PROGRAM P1_03_Alarms
VAR
	i					:USINT;
	bAlarmActive		:BOOL;
	bAlarmDisabled		:BOOL;
	TON_AlarmOK			:TON;

END_VAR
VAR PERSISTENT
	fbAlarm				:ARRAY [0..69] OF FB_AlarmDiagnostic;
END_VAR

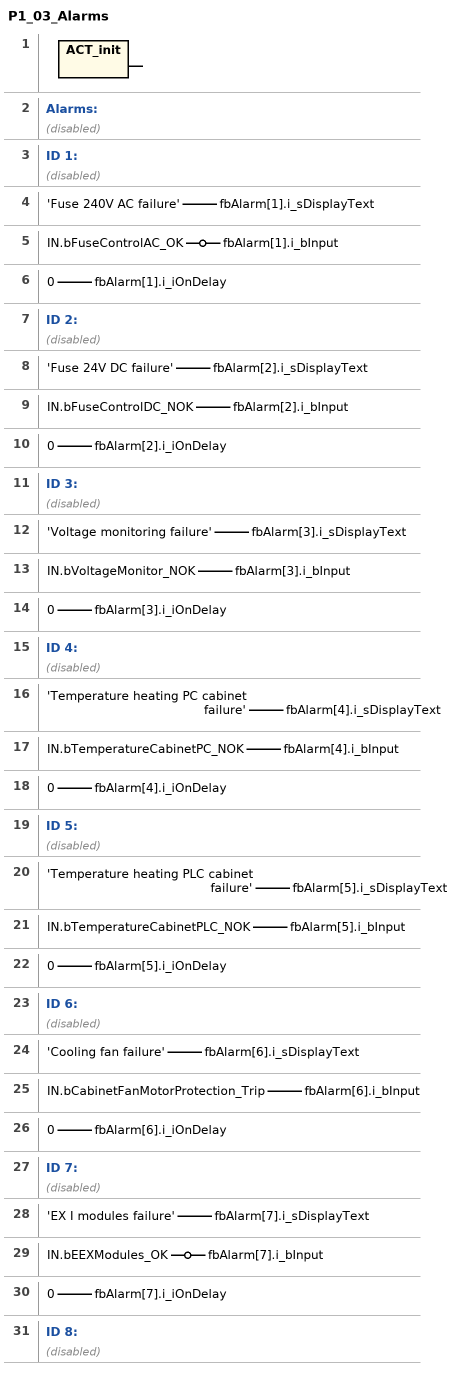
// NETWORK 1
ACT_init();

// NETWORK 2 (disabled)
// label: Alarms

// NETWORK 3 (disabled)
// label: ID 1

// NETWORK 4
fbAlarm[1].i_sDisplayText := 'Fuse 240V AC failure';

// NETWORK 5
fbAlarm[1].i_bInput := NOT IN.bFuseControlAC_OK;

// NETWORK 6
fbAlarm[1].i_iOnDelay := 0;

// NETWORK 7 (disabled)
// label: ID 2

// NETWORK 8
fbAlarm[2].i_sDisplayText := 'Fuse 24V DC failure';

// NETWORK 9
fbAlarm[2].i_bInput := IN.bFuseControlDC_NOK;

// NETWORK 10
fbAlarm[2].i_iOnDelay := 0;

// NETWORK 11 (disabled)
// label: ID 3

// NETWORK 12
fbAlarm[3].i_sDisplayText := 'Voltage monitoring failure';

// NETWORK 13
fbAlarm[3].i_bInput := IN.bVoltageMonitor_NOK;

// NETWORK 14
fbAlarm[3].i_iOnDelay := 0;

// NETWORK 15 (disabled)
// label: ID 4

// NETWORK 16
fbAlarm[4].i_sDisplayText := 'Temperature heating PC cabinet failure';

// NETWORK 17
fbAlarm[4].i_bInput := IN.bTemperatureCabinetPC_NOK;

// NETWORK 18
fbAlarm[4].i_iOnDelay := 0;

// NETWORK 19 (disabled)
// label: ID 5

// NETWORK 20
fbAlarm[5].i_sDisplayText := 'Temperature heating PLC cabinet failure';

// NETWORK 21
fbAlarm[5].i_bInput := IN.bTemperatureCabinetPLC_NOK;

// NETWORK 22
fbAlarm[5].i_iOnDelay := 0;

// NETWORK 23 (disabled)
// label: ID 6

// NETWORK 24
fbAlarm[6].i_sDisplayText := 'Cooling fan failure';

// NETWORK 25
fbAlarm[6].i_bInput := IN.bCabinetFanMotorProtection_Trip;

// NETWORK 26
fbAlarm[6].i_iOnDelay := 0;

// NETWORK 27 (disabled)
// label: ID 7

// NETWORK 28
fbAlarm[7].i_sDisplayText := 'EX I modules failure';

// NETWORK 29
fbAlarm[7].i_bInput := NOT IN.bEEXModules_OK;

// NETWORK 30
fbAlarm[7].i_iOnDelay := 0;

// NETWORK 31 (disabled)
// label: ID 8

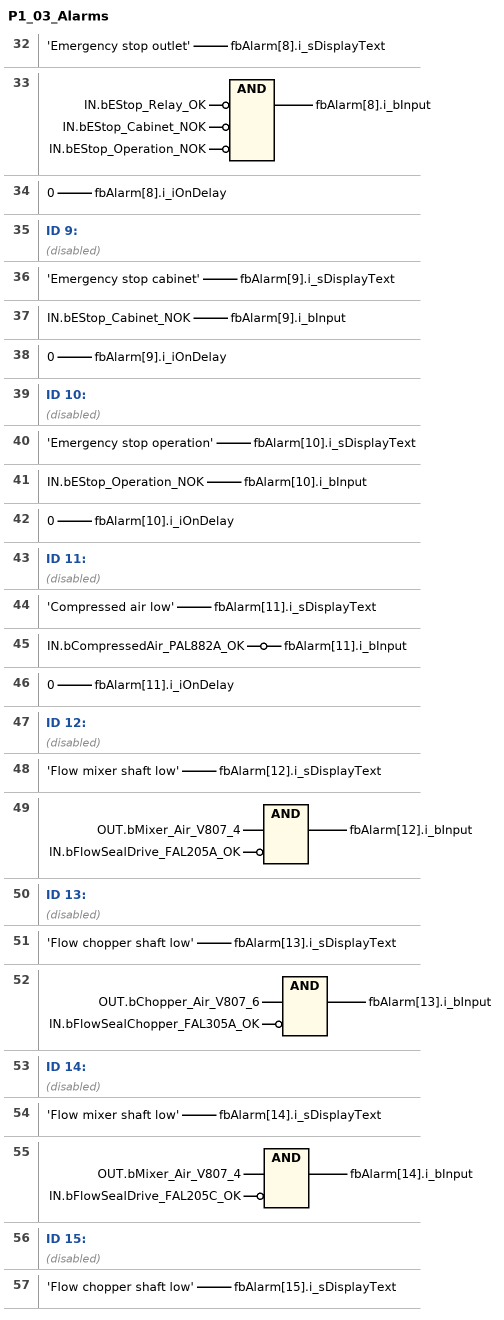
// NETWORK 32
fbAlarm[8].i_sDisplayText := 'Emergency stop outlet';

// NETWORK 33
fbAlarm[8].i_bInput := NOT IN.bEStop_Relay_OK AND NOT IN.bEStop_Cabinet_NOK AND NOT IN.bEStop_Operation_NOK;

// NETWORK 34
fbAlarm[8].i_iOnDelay := 0;

// NETWORK 35 (disabled)
// label: ID 9

// NETWORK 36
fbAlarm[9].i_sDisplayText := 'Emergency stop cabinet';

// NETWORK 37
fbAlarm[9].i_bInput := IN.bEStop_Cabinet_NOK;

// NETWORK 38
fbAlarm[9].i_iOnDelay := 0;

// NETWORK 39 (disabled)
// label: ID 10

// NETWORK 40
fbAlarm[10].i_sDisplayText := 'Emergency stop operation';

// NETWORK 41
fbAlarm[10].i_bInput := IN.bEStop_Operation_NOK;

// NETWORK 42
fbAlarm[10].i_iOnDelay := 0;

// NETWORK 43 (disabled)
// label: ID 11

// NETWORK 44
fbAlarm[11].i_sDisplayText := 'Compressed air low';

// NETWORK 45
fbAlarm[11].i_bInput := NOT IN.bCompressedAir_PAL882A_OK;

// NETWORK 46
fbAlarm[11].i_iOnDelay := 0;

// NETWORK 47 (disabled)
// label: ID 12

// NETWORK 48
fbAlarm[12].i_sDisplayText := 'Flow mixer shaft low';

// NETWORK 49
fbAlarm[12].i_bInput := OUT.bMixer_Air_V807_4 AND NOT IN.bFlowSealDrive_FAL205A_OK;

// NETWORK 50 (disabled)
// label: ID 13

// NETWORK 51
fbAlarm[13].i_sDisplayText := 'Flow chopper shaft low';

// NETWORK 52
fbAlarm[13].i_bInput := OUT.bChopper_Air_V807_6 AND NOT IN.bFlowSealChopper_FAL305A_OK;

// NETWORK 53 (disabled)
// label: ID 14

// NETWORK 54
fbAlarm[14].i_sDisplayText := 'Flow mixer shaft low';

// NETWORK 55
fbAlarm[14].i_bInput := OUT.bMixer_Air_V807_4 AND NOT IN.bFlowSealDrive_FAL205C_OK;

// NETWORK 56 (disabled)
// label: ID 15

// NETWORK 57
fbAlarm[15].i_sDisplayText := 'Flow chopper shaft low';

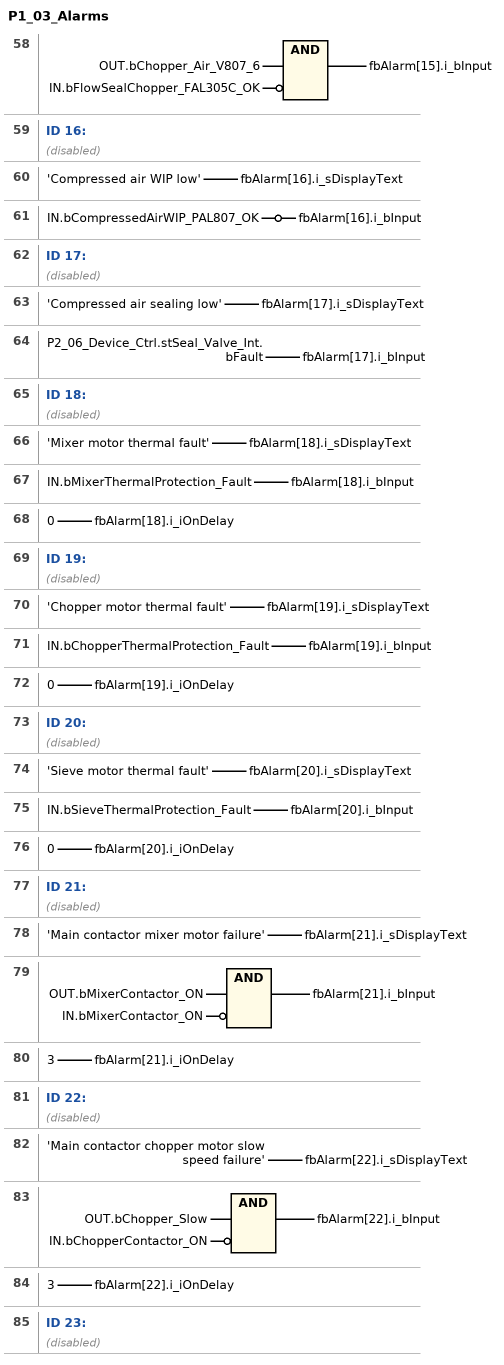
// NETWORK 58
fbAlarm[15].i_bInput := OUT.bChopper_Air_V807_6 AND NOT IN.bFlowSealChopper_FAL305C_OK;

// NETWORK 59 (disabled)
// label: ID 16

// NETWORK 60
fbAlarm[16].i_sDisplayText := 'Compressed air WIP low';

// NETWORK 61
fbAlarm[16].i_bInput := NOT IN.bCompressedAirWIP_PAL807_OK;

// NETWORK 62 (disabled)
// label: ID 17

// NETWORK 63
fbAlarm[17].i_sDisplayText := 'Compressed air sealing low';

// NETWORK 64
fbAlarm[17].i_bInput := P2_06_Device_Ctrl.stSeal_Valve_Int.bFault;

// NETWORK 65 (disabled)
// label: ID 18

// NETWORK 66
fbAlarm[18].i_sDisplayText := 'Mixer motor thermal fault';

// NETWORK 67
fbAlarm[18].i_bInput := IN.bMixerThermalProtection_Fault;

// NETWORK 68
fbAlarm[18].i_iOnDelay := 0;

// NETWORK 69 (disabled)
// label: ID 19

// NETWORK 70
fbAlarm[19].i_sDisplayText := 'Chopper motor thermal fault';

// NETWORK 71
fbAlarm[19].i_bInput := IN.bChopperThermalProtection_Fault;

// NETWORK 72
fbAlarm[19].i_iOnDelay := 0;

// NETWORK 73 (disabled)
// label: ID 20

// NETWORK 74
fbAlarm[20].i_sDisplayText := 'Sieve motor thermal fault';

// NETWORK 75
fbAlarm[20].i_bInput := IN.bSieveThermalProtection_Fault;

// NETWORK 76
fbAlarm[20].i_iOnDelay := 0;

// NETWORK 77 (disabled)
// label: ID 21

// NETWORK 78
fbAlarm[21].i_sDisplayText := 'Main contactor mixer motor failure';

// NETWORK 79
fbAlarm[21].i_bInput := OUT.bMixerContactor_ON AND NOT IN.bMixerContactor_ON;

// NETWORK 80
fbAlarm[21].i_iOnDelay := 3;

// NETWORK 81 (disabled)
// label: ID 22

// NETWORK 82
fbAlarm[22].i_sDisplayText := 'Main contactor chopper motor slow speed failure';

// NETWORK 83
fbAlarm[22].i_bInput := OUT.bChopper_Slow AND NOT IN.bChopperContactor_ON;

// NETWORK 84
fbAlarm[22].i_iOnDelay := 3;

// NETWORK 85 (disabled)
// label: ID 23

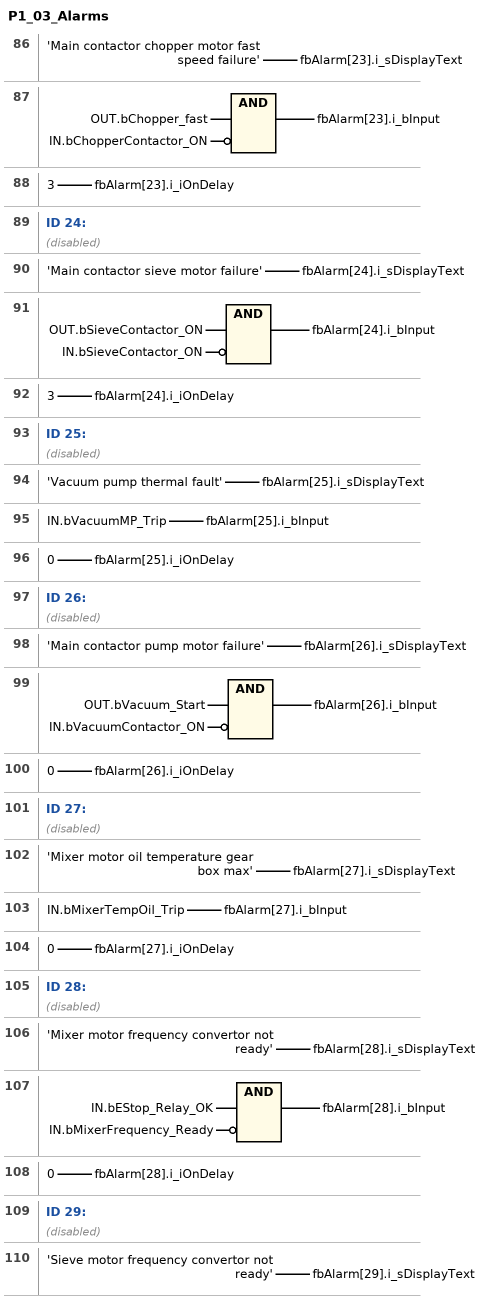
// NETWORK 86
fbAlarm[23].i_sDisplayText := 'Main contactor chopper motor fast speed failure';

// NETWORK 87
fbAlarm[23].i_bInput := OUT.bChopper_fast AND NOT IN.bChopperContactor_ON;

// NETWORK 88
fbAlarm[23].i_iOnDelay := 3;

// NETWORK 89 (disabled)
// label: ID 24

// NETWORK 90
fbAlarm[24].i_sDisplayText := 'Main contactor sieve motor failure';

// NETWORK 91
fbAlarm[24].i_bInput := OUT.bSieveContactor_ON AND NOT IN.bSieveContactor_ON;

// NETWORK 92
fbAlarm[24].i_iOnDelay := 3;

// NETWORK 93 (disabled)
// label: ID 25

// NETWORK 94
fbAlarm[25].i_sDisplayText := 'Vacuum pump thermal fault';

// NETWORK 95
fbAlarm[25].i_bInput := IN.bVacuumMP_Trip;

// NETWORK 96
fbAlarm[25].i_iOnDelay := 0;

// NETWORK 97 (disabled)
// label: ID 26

// NETWORK 98
fbAlarm[26].i_sDisplayText := 'Main contactor pump motor failure';

// NETWORK 99
fbAlarm[26].i_bInput := OUT.bVacuum_Start AND NOT IN.bVacuumContactor_ON;

// NETWORK 100
fbAlarm[26].i_iOnDelay := 0;

// NETWORK 101 (disabled)
// label: ID 27

// NETWORK 102
fbAlarm[27].i_sDisplayText := 'Mixer motor oil temperature gear box max';

// NETWORK 103
fbAlarm[27].i_bInput := IN.bMixerTempOil_Trip;

// NETWORK 104
fbAlarm[27].i_iOnDelay := 0;

// NETWORK 105 (disabled)
// label: ID 28

// NETWORK 106
fbAlarm[28].i_sDisplayText := 'Mixer motor frequency convertor not ready';

// NETWORK 107
fbAlarm[28].i_bInput := IN.bEStop_Relay_OK AND NOT IN.bMixerFrequency_Ready;

// NETWORK 108
fbAlarm[28].i_iOnDelay := 0;

// NETWORK 109 (disabled)
// label: ID 29

// NETWORK 110
fbAlarm[29].i_sDisplayText := 'Sieve motor frequency convertor not ready';

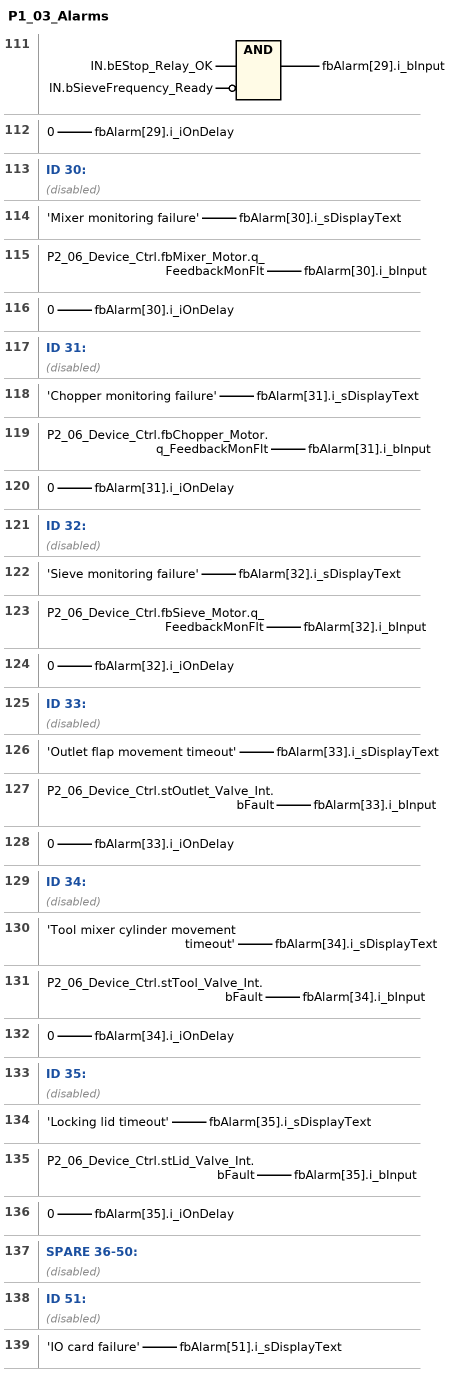
// NETWORK 111
fbAlarm[29].i_bInput := IN.bEStop_Relay_OK AND NOT IN.bSieveFrequency_Ready;

// NETWORK 112
fbAlarm[29].i_iOnDelay := 0;

// NETWORK 113 (disabled)
// label: ID 30

// NETWORK 114
fbAlarm[30].i_sDisplayText := 'Mixer monitoring failure';

// NETWORK 115
fbAlarm[30].i_bInput := P2_06_Device_Ctrl.fbMixer_Motor.q_FeedbackMonFlt;

// NETWORK 116
fbAlarm[30].i_iOnDelay := 0;

// NETWORK 117 (disabled)
// label: ID 31

// NETWORK 118
fbAlarm[31].i_sDisplayText := 'Chopper monitoring failure';

// NETWORK 119
fbAlarm[31].i_bInput := P2_06_Device_Ctrl.fbChopper_Motor.q_FeedbackMonFlt;

// NETWORK 120
fbAlarm[31].i_iOnDelay := 0;

// NETWORK 121 (disabled)
// label: ID 32

// NETWORK 122
fbAlarm[32].i_sDisplayText := 'Sieve monitoring failure';

// NETWORK 123
fbAlarm[32].i_bInput := P2_06_Device_Ctrl.fbSieve_Motor.q_FeedbackMonFlt;

// NETWORK 124
fbAlarm[32].i_iOnDelay := 0;

// NETWORK 125 (disabled)
// label: ID 33

// NETWORK 126
fbAlarm[33].i_sDisplayText := 'Outlet flap movement timeout';

// NETWORK 127
fbAlarm[33].i_bInput := P2_06_Device_Ctrl.stOutlet_Valve_Int.bFault;

// NETWORK 128
fbAlarm[33].i_iOnDelay := 0;

// NETWORK 129 (disabled)
// label: ID 34

// NETWORK 130
fbAlarm[34].i_sDisplayText := 'Tool mixer cylinder movement timeout';

// NETWORK 131
fbAlarm[34].i_bInput := P2_06_Device_Ctrl.stTool_Valve_Int.bFault;

// NETWORK 132
fbAlarm[34].i_iOnDelay := 0;

// NETWORK 133 (disabled)
// label: ID 35

// NETWORK 134
fbAlarm[35].i_sDisplayText := 'Locking lid timeout';

// NETWORK 135
fbAlarm[35].i_bInput := P2_06_Device_Ctrl.stLid_Valve_Int.bFault;

// NETWORK 136
fbAlarm[35].i_iOnDelay := 0;

// NETWORK 137 (disabled)
// label: SPARE 36-50

// NETWORK 138 (disabled)
// label: ID 51

// NETWORK 139
fbAlarm[51].i_sDisplayText := 'IO card failure';

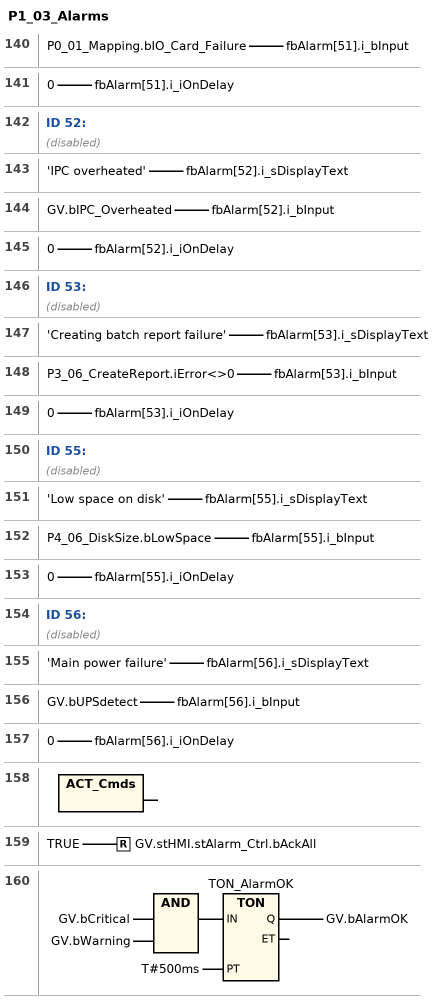
// NETWORK 140
fbAlarm[51].i_bInput := P0_01_Mapping.bIO_Card_Failure;

// NETWORK 141
fbAlarm[51].i_iOnDelay := 0;

// NETWORK 142 (disabled)
// label: ID 52

// NETWORK 143
fbAlarm[52].i_sDisplayText := 'IPC overheated';

// NETWORK 144
fbAlarm[52].i_bInput := GV.bIPC_Overheated;

// NETWORK 145
fbAlarm[52].i_iOnDelay := 0;

// NETWORK 146 (disabled)
// label: ID 53

// NETWORK 147
fbAlarm[53].i_sDisplayText := 'Creating batch report failure';

// NETWORK 148
fbAlarm[53].i_bInput := P3_06_CreateReport.iError<>0;

// NETWORK 149
fbAlarm[53].i_iOnDelay := 0;

// NETWORK 150 (disabled)
// label: ID 55

// NETWORK 151
fbAlarm[55].i_sDisplayText := 'Low space on disk';

// NETWORK 152
fbAlarm[55].i_bInput := P4_06_DiskSize.bLowSpace;

// NETWORK 153
fbAlarm[55].i_iOnDelay := 0;

// NETWORK 154 (disabled)
// label: ID 56

// NETWORK 155
fbAlarm[56].i_sDisplayText := 'Main power failure';

// NETWORK 156
fbAlarm[56].i_bInput := GV.bUPSdetect;

// NETWORK 157
fbAlarm[56].i_iOnDelay := 0;

// NETWORK 158
ACT_Cmds();

// NETWORK 159
GV.stHMI.stAlarm_Ctrl.bAckAll R= TRUE;

// NETWORK 160
TON_AlarmOK(IN := GV.bCritical AND GV.bWarning, PT := T#500ms); // TON
GV.bAlarmOK := TON_AlarmOK.Q;

ACTION ACT_Cmds:
GV.bCritical:=TRUE;
GV.bWarning:=TRUE;
bAlarmDisabled:=FALSE;
FOR i:=0 TO 50 DO
	//Init Function blocks
	fbAlarm[i](i_iID:=i,
			   i_bActive:=GV.stAlarm.Active[i],
			   q_bActive=>GV.stAlarm.Raise[i]);			
			   
	fbAlarm[i].i_bEnable:=TRUE;
	IF GV.stAlarm.Active[i] THEN
		IF i <= 25 THEN
			GV.bCritical:=FALSE;
		ELSIF i > 25 THEN
			GV.bWarning:=FALSE;
		END_IF
	END_IF
	
	//Raise
	IF GV.stAlarm.Raise[i] THEN
		GV.stAlarm.Alarm[i].Raise(0);
	END_IF
	
	//Active
	GV.stAlarm.Active[i]:=GV.stAlarm.Alarm[i].bActive;
	
	//Ack
	IF GV.stAlarm.Alarm[i].eConfirmationState = 3 OR GV.stHMI.stAlarm_Ctrl.bAckAll THEN
		GV.stAlarm.Alarm[i].Clear(0,1);
	END_IF
	
	//Clear warnings 
	IF GV.stAlarm.Active[i] AND NOT fbAlarm[i].i_bInput AND i>=25 THEN
		GV.stAlarm.Alarm[i].Clear(0,1);
	END_IF
	
	//Check disabled
	IF NOT fbAlarm[i].i_bEnable THEN
		bAlarmDisabled:=TRUE;
	END_IF
END_FOR
END_ACTION

ACTION ACT_Init:
IF MAIN.bFirstCycle THEN
	//Critical
	GV.stAlarm.Alarm[1].CreateEx(TC_EVENTS.Alarms.AlarmsEvent1,1,0);
	GV.stAlarm.Alarm[2].CreateEx(TC_EVENTS.Alarms.AlarmsEvent2,1,0);
	GV.stAlarm.Alarm[3].CreateEx(TC_EVENTS.Alarms.AlarmsEvent3,1,0);
	GV.stAlarm.Alarm[4].CreateEx(TC_EVENTS.Alarms.AlarmsEvent4,1,0);
	GV.stAlarm.Alarm[5].CreateEx(TC_EVENTS.Alarms.AlarmsEvent5,1,0);
	GV.stAlarm.Alarm[6].CreateEx(TC_EVENTS.Alarms.AlarmsEvent6,1,0);
	GV.stAlarm.Alarm[7].CreateEx(TC_EVENTS.Alarms.AlarmsEvent7,1,0);
	GV.stAlarm.Alarm[8].CreateEx(TC_EVENTS.Alarms.AlarmsEvent8,1,0);
	GV.stAlarm.Alarm[9].CreateEx(TC_EVENTS.Alarms.AlarmsEvent9,1,0);
	GV.stAlarm.Alarm[10].CreateEx(TC_EVENTS.Alarms.AlarmsEvent10,1,0);
	GV.stAlarm.Alarm[11].CreateEx(TC_EVENTS.Alarms.AlarmsEvent11,1,0);
	GV.stAlarm.Alarm[12].CreateEx(TC_EVENTS.Alarms.AlarmsEvent12,1,0);
	GV.stAlarm.Alarm[13].CreateEx(TC_EVENTS.Alarms.AlarmsEvent13,1,0);
	GV.stAlarm.Alarm[14].CreateEx(TC_EVENTS.Alarms.AlarmsEvent14,1,0);
	GV.stAlarm.Alarm[15].CreateEx(TC_EVENTS.Alarms.AlarmsEvent15,1,0);
	GV.stAlarm.Alarm[16].CreateEx(TC_EVENTS.Alarms.AlarmsEvent16,1,0);
	GV.stAlarm.Alarm[17].CreateEx(TC_EVENTS.Alarms.AlarmsEvent17,1,0);
	GV.stAlarm.Alarm[18].CreateEx(TC_EVENTS.Alarms.AlarmsEvent18,1,0);
	GV.stAlarm.Alarm[19].CreateEx(TC_EVENTS.Alarms.AlarmsEvent19,1,0);
	GV.stAlarm.Alarm[20].CreateEx(TC_EVENTS.Alarms.AlarmsEvent20,1,0);
	GV.stAlarm.Alarm[21].CreateEx(TC_EVENTS.Alarms.AlarmsEvent21,1,0);
	GV.stAlarm.Alarm[22].CreateEx(TC_EVENTS.Alarms.AlarmsEvent22,1,0);
	GV.stAlarm.Alarm[23].CreateEx(TC_EVENTS.Alarms.AlarmsEvent23,1,0);
	GV.stAlarm.Alarm[24].CreateEx(TC_EVENTS.Alarms.AlarmsEvent24,1,0);
	GV.stAlarm.Alarm[25].CreateEx(TC_EVENTS.Alarms.AlarmsEvent25,1,0);
	GV.stAlarm.Alarm[26].CreateEx(TC_EVENTS.Alarms.AlarmsEvent26,1,0);
	GV.stAlarm.Alarm[27].CreateEx(TC_EVENTS.Alarms.AlarmsEvent27,1,0);
	GV.stAlarm.Alarm[28].CreateEx(TC_EVENTS.Alarms.AlarmsEvent28,1,0);
	GV.stAlarm.Alarm[29].CreateEx(TC_EVENTS.Alarms.AlarmsEvent29,1,0);
	GV.stAlarm.Alarm[30].CreateEx(TC_EVENTS.Alarms.AlarmsEvent30,1,0);
	GV.stAlarm.Alarm[31].CreateEx(TC_EVENTS.Alarms.AlarmsEvent31,1,0);
	GV.stAlarm.Alarm[32].CreateEx(TC_EVENTS.Alarms.AlarmsEvent32,1,0);
	GV.stAlarm.Alarm[33].CreateEx(TC_EVENTS.Alarms.AlarmsEvent33,1,0);
	GV.stAlarm.Alarm[34].CreateEx(TC_EVENTS.Alarms.AlarmsEvent34,1,0);
	GV.stAlarm.Alarm[35].CreateEx(TC_EVENTS.Alarms.AlarmsEvent35,1,0);
	GV.stAlarm.Alarm[36].CreateEx(TC_EVENTS.Alarms.AlarmsEvent36,1,0);
	GV.stAlarm.Alarm[37].CreateEx(TC_EVENTS.Alarms.AlarmsEvent37,1,0);
	GV.stAlarm.Alarm[38].CreateEx(TC_EVENTS.Alarms.AlarmsEvent38,1,0);
	GV.stAlarm.Alarm[39].CreateEx(TC_EVENTS.Alarms.AlarmsEvent39,1,0);
	GV.stAlarm.Alarm[40].CreateEx(TC_EVENTS.Alarms.AlarmsEvent40,1,0);	
	GV.stAlarm.Alarm[41].CreateEx(TC_EVENTS.Alarms.AlarmsEvent41,1,0);
	GV.stAlarm.Alarm[42].CreateEx(TC_EVENTS.Alarms.AlarmsEvent42,1,0);
	GV.stAlarm.Alarm[43].CreateEx(TC_EVENTS.Alarms.AlarmsEvent43,1,0);
	GV.stAlarm.Alarm[44].CreateEx(TC_EVENTS.Alarms.AlarmsEvent44,1,0);
	GV.stAlarm.Alarm[45].CreateEx(TC_EVENTS.Alarms.AlarmsEvent45,1,0);
	GV.stAlarm.Alarm[46].CreateEx(TC_EVENTS.Alarms.AlarmsEvent46,1,0);
	GV.stAlarm.Alarm[47].CreateEx(TC_EVENTS.Alarms.AlarmsEvent47,1,0);
	GV.stAlarm.Alarm[48].CreateEx(TC_EVENTS.Alarms.AlarmsEvent48,1,0);
	GV.stAlarm.Alarm[49].CreateEx(TC_EVENTS.Alarms.AlarmsEvent49,1,0);
	GV.stAlarm.Alarm[50].CreateEx(TC_EVENTS.Alarms.AlarmsEvent50,1,0);
	GV.stAlarm.Alarm[51].CreateEx(TC_EVENTS.Alarms.AlarmsEvent51,1,0);
	GV.stAlarm.Alarm[52].CreateEx(TC_EVENTS.Alarms.AlarmsEvent52,1,0);
	GV.stAlarm.Alarm[53].CreateEx(TC_EVENTS.Alarms.AlarmsEvent53,1,0);
	GV.stAlarm.Alarm[54].CreateEx(TC_EVENTS.Alarms.AlarmsEvent54,1,0);
	GV.stAlarm.Alarm[55].CreateEx(TC_EVENTS.Alarms.AlarmsEvent55,1,0);
	GV.stAlarm.Alarm[56].CreateEx(TC_EVENTS.Alarms.AlarmsEvent56,1,0);
	GV.stAlarm.Alarm[57].CreateEx(TC_EVENTS.Alarms.AlarmsEvent57,1,0);
	GV.stAlarm.Alarm[58].CreateEx(TC_EVENTS.Alarms.AlarmsEvent58,1,0);
	GV.stAlarm.Alarm[59].CreateEx(TC_EVENTS.Alarms.AlarmsEvent59,1,0);
	GV.stAlarm.Alarm[60].CreateEx(TC_EVENTS.Alarms.AlarmsEvent60,1,0);
	//SP
	GV.stAlarm.Alarm[61].CreateEx(TC_EVENTS.Alarms.AlarmsEvent61,1,0);
	GV.stAlarm.Alarm[62].CreateEx(TC_EVENTS.Alarms.AlarmsEvent62,1,0);
	GV.stAlarm.Alarm[63].CreateEx(TC_EVENTS.Alarms.AlarmsEvent63,1,0);
	GV.stAlarm.Alarm[64].CreateEx(TC_EVENTS.Alarms.AlarmsEvent64,1,0);
	GV.stAlarm.Alarm[65].CreateEx(TC_EVENTS.Alarms.AlarmsEvent65,1,0);
	GV.stAlarm.Alarm[66].CreateEx(TC_EVENTS.Alarms.AlarmsEvent66,1,0);
	GV.stAlarm.Alarm[67].CreateEx(TC_EVENTS.Alarms.AlarmsEvent67,1,0);
	GV.stAlarm.Alarm[68].CreateEx(TC_EVENTS.Alarms.AlarmsEvent68,1,0);
	GV.stAlarm.Alarm[69].CreateEx(TC_EVENTS.Alarms.AlarmsEvent69,1,0);
	GV.stAlarm.Alarm[70].CreateEx(TC_EVENTS.Alarms.AlarmsEvent70,1,0);
END_IF
END_ACTION

END_PROGRAM

(* stored: Version 1.1.0.1, ProductVersion 3.1.4026.13
   POU P1_03_Alarms: Id {5dbba99e-5643-4941-9e20-3c5bab16130f}, SpecialFunc None
   Action ACT_Cmds: Id {71f031f1-f00f-4b95-bee0-593fbbc853bd}
   Action ACT_Init: Id {a64be506-037f-4f62-9e07-bad88d9e4387} *)
